FUNCTION_BLOCK FLOOR_Test EXTENDS FB_TestSuite
VAR_INPUT
END_VAR
VAR_OUTPUT
END_VAR
VAR
END_VAR

PositivePieToThree();
NegativePieToNegativeFour();
TwoToTwo();

METHOD NegativePieToNegativeFour
VAR
	Result : INT;
	ExpectedFloor : INT := -4;
END_VAR
TEST('NegativePieToNegativeFour');
 
Result := FLOOR(X := -3.14);
 
AssertEquals(Expected := ExpectedFloor,
             Actual := Result,
             Message := 'The calculation is not correct');
 
TEST_FINISHED();
END_METHOD

METHOD PositivePieToThree
VAR
	Result : INT;
	ExpectedFloor : INT := 3;
END_VAR
TEST('PositivePieToThree');
 
Result := FLOOR(X := 3.14);
 
AssertEquals(Expected := ExpectedFloor,
             Actual := Result,
             Message := 'The calculation is not correct');
 
TEST_FINISHED();
END_METHOD

METHOD TwoToTwo
VAR
	Result : INT;
	ExpectedFloor : INT := 2;
END_VAR
TEST('TwoToTwo');
 
Result := FLOOR(X := 2);
 
AssertEquals(Expected := ExpectedFloor,
             Actual := Result,
             Message := 'The calculation is not correct');
 
TEST_FINISHED();
END_METHOD

END_FUNCTION_BLOCK

(* stored: Version 1.1.0.1, ProductVersion 3.1.4024.9
   POU FLOOR_Test: Id {076c40d4-c709-4804-a456-c2b292fdb9ad}, SpecialFunc None
   Method NegativePieToNegativeFour: Id {f38383cb-b87e-4315-8d22-909e3d3c9184}
   Method PositivePieToThree: Id {d3a835b1-322e-4b48-b2e6-a6731a35a8fd}
   Method TwoToTwo: Id {845fdea8-ebbd-487d-bde5-1b2cc49bcb4d} *)
